Fanuc KAREL source: kt00220.KL

-- PROVISIONAL review KL for V940-1; original PC SHA256 6f4de5b31bdc2251faf18d05ceffd3b4169192aae48d265d38b6c434b029d20a
-- Incomplete behavior may be omitted. Consult companion uncertainty JSON. Do not deploy.
PROGRAM KT00220
%NOLOCKGROUP
VAR
  I2 : INTEGER
  OUT : INTEGER
-- UNRESOLVED_DECL H1 type=002017
BEGIN
  -- V9_ZERO_TABLE_METADATA_HINT layout=0001; no indexed target words; source/name/runtime held
  -- UNRESOLVED_PC offsets 5-19; opcodes 2E,22,9D,33,B4
  -- UNRESOLVED_PC offsets 24-35; opcodes 2E,23
  -- UNRESOLVED_PC offsets 40-62; opcodes 22,9D,33,B3,21,46,23
  -- UNRESOLVED_PC offsets 67-71; opcodes 7F
END KT00220
